(* IEC 61131-3 sources: AOI-sys-for-TI/src/plc, 3 files *)

(* ---- safety_program.st ---- *)
(* ==========================================================================
 * Program:     SAFETY_PROGRAM
 * Description: Safety PLC Logic for AOI Inspection System
 * Target:      Mitsubishi iQ-R Safety CPU (R6SFM)
 * Standard:    ISO 13849-1 PLd, Category 3 (dual-channel with diagnostics)
 *              IEC 62061 SIL 2
 * Notes:       All safety-related I/O uses dual-channel cross-monitoring.
 *              Diagnostic coverage (DC) >= 90% per ISO 13849-1 Table D.2.
 *              CC-Link IE Field Safety protocol for distributed safety I/O.
 * ========================================================================== *)

SAFETY_PROGRAM SAFETY_MAIN

(* ---- Safety I/O Type Definitions ---------------------------------------- *)
TYPE ST_DUAL_CHANNEL : STRUCT
    CH_A             : BOOL;          (* Primary channel input *)
    CH_B             : BOOL;          (* Redundant channel input *)
    DISCREPANCY      : BOOL;          (* Cross-monitor fault detected *)
    DISC_TIMER       : TON;           (* Discrepancy time window *)
    VALID            : BOOL;          (* Both channels agree and healthy *)
END_STRUCT;
END_TYPE

TYPE ST_LIGHT_CURTAIN : STRUCT
    OSSD_1           : BOOL;          (* IEC 61496 Type 2 output 1 *)
    OSSD_2           : BOOL;          (* Redundant safety output 2 *)
    MUTING_ACTIVE    : BOOL;          (* Muting lamp + bypass engaged *)
    BLANKING_ZONE    : USINT;         (* Fixed blanking for material passage *)
    FAULT            : BOOL;
END_STRUCT;
END_TYPE

(* ---- Safety Variables --------------------------------------------------- *)
VAR
    (* E-Stop circuits: 3 buttons per ISO 13850 (twist-release, red/yellow) *)
    ESTOP_1          : ST_DUAL_CHANNEL;   (* Main operator panel *)
    ESTOP_2          : ST_DUAL_CHANNEL;   (* Rear access panel *)
    ESTOP_3          : ST_DUAL_CHANNEL;   (* Teach pendant / mobile *)

    (* Light curtains: IEC 61496 Type 2, 14mm resolution *)
    LC_LOAD_ZONE     : ST_LIGHT_CURTAIN;  (* Loading side *)
    LC_UNLOAD_ZONE   : ST_LIGHT_CURTAIN;  (* Unloading side *)

    (* Safety door interlocks: tongue-type with solenoid lock *)
    DOOR_FRONT       : ST_DUAL_CHANNEL;   (* Front maintenance door *)
    DOOR_REAR        : ST_DUAL_CHANNEL;   (* Rear access door *)
    DOOR_LOCK_FRONT  : BOOL;              (* Solenoid lock output *)
    DOOR_LOCK_REAR   : BOOL;              (* Solenoid lock output *)

    (* Safe Torque Off contactors for servo drives *)
    STO_CONTACTOR_1  : BOOL;              (* Axes 1-4 group *)
    STO_CONTACTOR_2  : BOOL;              (* Axes 5-8 group *)
    STO_FEEDBACK_1   : ST_DUAL_CHANNEL;   (* Contactor weld-check via NC aux *)
    STO_FEEDBACK_2   : ST_DUAL_CHANNEL;

    (* Muting sensors for automatic material handling *)
    MUTE_SENSOR_1    : BOOL;              (* Entry photoeye - conveyor infeed *)
    MUTE_SENSOR_2    : BOOL;              (* Exit photoeye - conveyor infeed *)
    MUTE_SENSOR_3    : BOOL;              (* Entry photoeye - conveyor outfeed *)
    MUTE_SENSOR_4    : BOOL;              (* Exit photoeye - conveyor outfeed *)
    MUTE_TIMER_LOAD  : TON;
    MUTE_TIMER_UNLOAD: TON;

    (* Aggregate outputs *)
    SAFETY_RELAY_OK  : BOOL;              (* Master safety output to main PLC *)
    SAFETY_FAULT_CODE: WORD := 0;
    SAFETY_RESET_PB  : BOOL;              (* Manual reset required after fault *)
    RT_SAFETY_RESET  : R_TRIG;

    (* Discrepancy timing *)
    T_DISC_WINDOW    : TIME := T#500ms;   (* Max allowed discrepancy per Cat.3 *)
    T_MUTE_MAX       : TIME := T#10s;     (* Muting timeout: prevents stuck mute *)

    (* Diagnostic counters -- written to safety log every power cycle *)
    DIAG_ESTOP_TRIPS      : UDINT;
    DIAG_LC_INTERRUPTIONS : UDINT;
    DIAG_DOOR_FAULTS      : UDINT;
    DIAG_DISC_FAULTS      : UDINT;
END_VAR

(* ======================================================================== *)
(* DUAL-CHANNEL CROSS-MONITORING FUNCTION                                   *)
(* Category 3 requires detection of single faults. Discrepancy between      *)
(* channel A and B within T_DISC_WINDOW indicates wiring fault or contact   *)
(* welding. DC >= 90% achieved through cross-monitoring + watchdog.         *)
(* ======================================================================== *)

(* --- E-Stop 1: Main panel ----------------------------------------------- *)
ESTOP_1.DISC_TIMER(IN := (ESTOP_1.CH_A XOR ESTOP_1.CH_B), PT := T_DISC_WINDOW);
ESTOP_1.DISCREPANCY := ESTOP_1.DISC_TIMER.Q;
ESTOP_1.VALID := ESTOP_1.CH_A AND ESTOP_1.CH_B AND NOT ESTOP_1.DISCREPANCY;

(* --- E-Stop 2: Rear panel ----------------------------------------------- *)
ESTOP_2.DISC_TIMER(IN := (ESTOP_2.CH_A XOR ESTOP_2.CH_B), PT := T_DISC_WINDOW);
ESTOP_2.DISCREPANCY := ESTOP_2.DISC_TIMER.Q;
ESTOP_2.VALID := ESTOP_2.CH_A AND ESTOP_2.CH_B AND NOT ESTOP_2.DISCREPANCY;

(* --- E-Stop 3: Mobile / teach pendant ----------------------------------- *)
ESTOP_3.DISC_TIMER(IN := (ESTOP_3.CH_A XOR ESTOP_3.CH_B), PT := T_DISC_WINDOW);
ESTOP_3.DISCREPANCY := ESTOP_3.DISC_TIMER.Q;
ESTOP_3.VALID := ESTOP_3.CH_A AND ESTOP_3.CH_B AND NOT ESTOP_3.DISCREPANCY;

(* --- Light curtain monitoring ------------------------------------------- *)
(* IEC 61496 Type 2: OSSD outputs are antivalent pulsed; both must be TRUE
   for safe condition. Internal diagnostics handled by curtain controller. *)
LC_LOAD_ZONE.FAULT   := (LC_LOAD_ZONE.OSSD_1 XOR LC_LOAD_ZONE.OSSD_2);
LC_UNLOAD_ZONE.FAULT := (LC_UNLOAD_ZONE.OSSD_1 XOR LC_UNLOAD_ZONE.OSSD_2);

(* --- Muting logic for load zone ----------------------------------------- *)
(* Muting allows automatic material (basket/magazine) to pass through the
   light curtain without triggering a safety stop. Sequential activation
   of two cross-beam sensors validates material presence vs. operator.    *)
IF MUTE_SENSOR_1 AND MUTE_SENSOR_2 AND NOT LC_LOAD_ZONE.FAULT THEN
    LC_LOAD_ZONE.MUTING_ACTIVE := TRUE;
    MUTE_TIMER_LOAD(IN := TRUE, PT := T_MUTE_MAX);
ELSE
    IF NOT MUTE_SENSOR_1 AND NOT MUTE_SENSOR_2 THEN
        LC_LOAD_ZONE.MUTING_ACTIVE := FALSE;
        MUTE_TIMER_LOAD(IN := FALSE);
    END_IF;
END_IF;

(* Muting timeout: if material jams, revert to protected mode *)
IF MUTE_TIMER_LOAD.Q THEN
    LC_LOAD_ZONE.MUTING_ACTIVE := FALSE;
    MUTE_TIMER_LOAD(IN := FALSE);
    SAFETY_FAULT_CODE := 16#5001;  (* Muting timeout - check conveyor jam *)
END_IF;

(* --- Muting logic for unload zone --------------------------------------- *)
IF MUTE_SENSOR_3 AND MUTE_SENSOR_4 AND NOT LC_UNLOAD_ZONE.FAULT THEN
    LC_UNLOAD_ZONE.MUTING_ACTIVE := TRUE;
    MUTE_TIMER_UNLOAD(IN := TRUE, PT := T_MUTE_MAX);
ELSE
    IF NOT MUTE_SENSOR_3 AND NOT MUTE_SENSOR_4 THEN
        LC_UNLOAD_ZONE.MUTING_ACTIVE := FALSE;
        MUTE_TIMER_UNLOAD(IN := FALSE);
    END_IF;
END_IF;

IF MUTE_TIMER_UNLOAD.Q THEN
    LC_UNLOAD_ZONE.MUTING_ACTIVE := FALSE;
    MUTE_TIMER_UNLOAD(IN := FALSE);
    SAFETY_FAULT_CODE := 16#5002;
END_IF;

(* --- Safety door interlock monitoring ----------------------------------- *)
DOOR_FRONT.DISC_TIMER(IN := (DOOR_FRONT.CH_A XOR DOOR_FRONT.CH_B), PT := T_DISC_WINDOW);
DOOR_FRONT.DISCREPANCY := DOOR_FRONT.DISC_TIMER.Q;
DOOR_FRONT.VALID := DOOR_FRONT.CH_A AND DOOR_FRONT.CH_B AND NOT DOOR_FRONT.DISCREPANCY;

DOOR_REAR.DISC_TIMER(IN := (DOOR_REAR.CH_A XOR DOOR_REAR.CH_B), PT := T_DISC_WINDOW);
DOOR_REAR.DISCREPANCY := DOOR_REAR.DISC_TIMER.Q;
DOOR_REAR.VALID := DOOR_REAR.CH_A AND DOOR_REAR.CH_B AND NOT DOOR_REAR.DISCREPANCY;

(* Solenoid door locks: keep locked when machine running, unlock on safe stop *)
DOOR_LOCK_FRONT := SAFETY_RELAY_OK;
DOOR_LOCK_REAR  := SAFETY_RELAY_OK;

(* --- STO contactor feedback monitoring ---------------------------------- *)
(* NC auxiliary contacts on STO contactors provide weld-detection.
   If contactor is commanded OFF but feedback shows still ON, weld fault. *)
STO_FEEDBACK_1.DISC_TIMER(IN := (STO_FEEDBACK_1.CH_A XOR STO_FEEDBACK_1.CH_B), PT := T_DISC_WINDOW);
STO_FEEDBACK_1.DISCREPANCY := STO_FEEDBACK_1.DISC_TIMER.Q;
STO_FEEDBACK_1.VALID := STO_FEEDBACK_1.CH_A AND STO_FEEDBACK_1.CH_B AND NOT STO_FEEDBACK_1.DISCREPANCY;

STO_FEEDBACK_2.DISC_TIMER(IN := (STO_FEEDBACK_2.CH_A XOR STO_FEEDBACK_2.CH_B), PT := T_DISC_WINDOW);
STO_FEEDBACK_2.DISCREPANCY := STO_FEEDBACK_2.DISC_TIMER.Q;
STO_FEEDBACK_2.VALID := STO_FEEDBACK_2.CH_A AND STO_FEEDBACK_2.CH_B AND NOT STO_FEEDBACK_2.DISCREPANCY;

(* ======================================================================== *)
(* MASTER SAFETY OUTPUT EVALUATION                                          *)
(* All conditions must be TRUE for machine to operate.                      *)
(* Any single failure -> immediate safe state (STO + pneumatic exhaust).    *)
(*                                                                          *)
(* Diagnostic Coverage Calculation (ISO 13849-1 Table D.4):                 *)
(*   E-Stop dual-channel cross-monitored:        DC = 99%                  *)
(*   Light curtain Type 2 + muting:              DC = 90%                  *)
(*   Safety door interlock dual-channel:         DC = 99%                  *)
(*   STO contactor with weld-check feedback:     DC = 99%                  *)
(*   Overall DC_avg >= 90% -> meets Cat.3 PLd requirement                  *)
(*                                                                          *)
(*   MTTFd per channel > 30 years (high reliability components)            *)
(*   CCF score >= 65 points (separate routing, different manufacturers)     *)
(* ======================================================================== *)

SAFETY_RELAY_OK :=
    ESTOP_1.VALID AND
    ESTOP_2.VALID AND
    ESTOP_3.VALID AND
    DOOR_FRONT.VALID AND
    DOOR_REAR.VALID AND
    (LC_LOAD_ZONE.OSSD_1 AND LC_LOAD_ZONE.OSSD_2 OR LC_LOAD_ZONE.MUTING_ACTIVE) AND
    (LC_UNLOAD_ZONE.OSSD_1 AND LC_UNLOAD_ZONE.OSSD_2 OR LC_UNLOAD_ZONE.MUTING_ACTIVE) AND
    NOT LC_LOAD_ZONE.FAULT AND
    NOT LC_UNLOAD_ZONE.FAULT AND
    STO_FEEDBACK_1.VALID AND
    STO_FEEDBACK_2.VALID AND
    (SAFETY_FAULT_CODE = 0);

(* --- STO contactor control ---------------------------------------------- *)
(* Energise STO contactors only when safety chain is healthy *)
STO_CONTACTOR_1 := SAFETY_RELAY_OK;
STO_CONTACTOR_2 := SAFETY_RELAY_OK;

(* --- Discrepancy fault latching ----------------------------------------- *)
(* Any discrepancy is latched until manual reset per ISO 13849-1 Cat.3     *)
IF ESTOP_1.DISCREPANCY OR ESTOP_2.DISCREPANCY OR ESTOP_3.DISCREPANCY THEN
    SAFETY_FAULT_CODE := 16#E100;  (* E-Stop discrepancy - check wiring *)
    DIAG_DISC_FAULTS := DIAG_DISC_FAULTS + 1;
END_IF;

IF DOOR_FRONT.DISCREPANCY OR DOOR_REAR.DISCREPANCY THEN
    SAFETY_FAULT_CODE := 16#E200;  (* Door interlock discrepancy *)
    DIAG_DOOR_FAULTS := DIAG_DOOR_FAULTS + 1;
END_IF;

IF STO_FEEDBACK_1.DISCREPANCY OR STO_FEEDBACK_2.DISCREPANCY THEN
    SAFETY_FAULT_CODE := 16#E300;  (* STO contactor weld detected *)
    DIAG_DISC_FAULTS := DIAG_DISC_FAULTS + 1;
END_IF;

(* --- Manual reset logic ------------------------------------------------- *)
(* ISO 13849-1 requires monitored manual reset after any safety event.
   Reset button must be outside the hazardous zone.                        *)
RT_SAFETY_RESET(CLK := SAFETY_RESET_PB);
IF RT_SAFETY_RESET.Q THEN
    (* Only allow reset if all physical inputs are in safe state *)
    IF ESTOP_1.CH_A AND ESTOP_1.CH_B AND
       ESTOP_2.CH_A AND ESTOP_2.CH_B AND
       ESTOP_3.CH_A AND ESTOP_3.CH_B AND
       DOOR_FRONT.CH_A AND DOOR_FRONT.CH_B AND
       DOOR_REAR.CH_A AND DOOR_REAR.CH_B THEN
        SAFETY_FAULT_CODE := 0;
    END_IF;
END_IF;

END_PROGRAM

(* ---- main_sequence.st ---- *)
(* =============================================================================
 * Program:     MAIN_SEQUENCE
 * Project:     TI AOI Inspection System
 * Controller:  Mitsubishi iQ-R Series (R16CPU + RJ71GF11-T2)
 * Network:     CC-Link IE Field Basic 1 Gbps (servo + remote I/O)
 *              EtherNet/IP CIP (IPC vision host communication)
 * Cycle Time:  0.5 ms fixed scan | 3.8 s total throughput (4-unit batch)
 * Author:      Controls Engineering
 * Revision:    1.0
 * ========================================================================== *)

PROGRAM MAIN_SEQUENCE

(* ---------------------------------------------------------------------------
 * TYPE DEFINITIONS
 * ------------------------------------------------------------------------ *)
TYPE
    E_INSPECT_STATE : (
        ST_IDLE             := 0,
        ST_BASKET_FEED      := 1,
        ST_CSE_LOAD         := 2,
        ST_PITCH_CHANGE     := 3,
        ST_TRANSFER_1       := 4,
        ST_TRANSFER_2       := 5,
        ST_TRANSFER_3       := 6,
        ST_TRANSFER_4       := 7,
        ST_TRANSFER_5       := 8,
        ST_TRANSFER_6       := 9,
        ST_CCD4_CHECK       := 10,  (* Bottom inspection - inverted optics *)
        ST_CCD3_CHECK       := 11,  (* Top surface inspection *)
        ST_CCD1_CHECK       := 12,  (* Side A + marking verification *)
        ST_ORIENT_COMP      := 13,  (* Theta correction from CCD1 result *)
        ST_CCD2_CHECK       := 14,  (* Side B after orientation alignment *)
        ST_UNLOAD_OK        := 15,
        ST_NG_SORT          := 16,  (* Divert to NG bin by defect class *)
        ST_NG_UNLOAD        := 17,
        ST_ERROR            := 99
    );

    TYPE_VISION_RESULT : STRUCT
        JUDGE           : BOOL;     (* TRUE = PASS, FALSE = NG *)
        DEFECT_CODE     : INT;      (* 0=OK, 1=scratch, 2=chip, 3=mark, 4=foreign *)
        OFFSET_X        : REAL;     (* um, positional deviation *)
        OFFSET_Y        : REAL;
        OFFSET_THETA    : REAL;     (* degrees, rotation deviation *)
        INSPECT_TIME_MS : INT;      (* Vision processing elapsed time *)
    END_STRUCT;

    TYPE_AXIS_CMD : STRUCT
        TARGET_POS      : DINT;     (* Command position in encoder pulses *)
        SPEED           : DINT;     (* mm/s x 100 for fixed-point *)
        ACCEL           : DINT;     (* mm/s^2 x 100 *)
        DECEL           : DINT;
        IN_POSITION     : BOOL;     (* Servo positioning complete feedback *)
        BUSY            : BOOL;
        ERROR           : BOOL;
    END_STRUCT;
END_TYPE

(* ---------------------------------------------------------------------------
 * VARIABLE DECLARATIONS
 * ------------------------------------------------------------------------ *)
VAR
    (* State machine *)
    CURRENT_STATE       : E_INSPECT_STATE := ST_IDLE;
    NEXT_STATE          : E_INSPECT_STATE;
    STATE_ENTRY         : BOOL := TRUE;         (* One-shot on state entry *)
    STEP_TIMER          : TON;                  (* Timeout watchdog per step *)
    CYCLE_TIMER         : TON;                  (* Total cycle time monitor *)
    STEP_TIMEOUT_MS     : TIME := T#5000ms;     (* Max dwell per state *)

    (* CC-Link IE Field cyclic I/O - 8 servo axes *)
    AXIS              : ARRAY[1..8] OF TYPE_AXIS_CMD;
    (* Axis mapping:
       1 = Transfer 1 (basket to pitch change)
       2 = Transfer 2 (pitch change to CCD4)
       3 = Transfer 3 (CCD4 to CCD3)
       4 = Transfer 4 (CCD3 to CCD1)
       5 = Transfer 5 (CCD1 to orient/CCD2)
       6 = Transfer 6 (orient/CCD2 to unload)
       7 = Orientation compensation theta axis
       8 = Side check rotation axis *)

    (* Vision handshake signals - EtherNet/IP CIP implicit messaging *)
    VISION_TRIG         : ARRAY[1..4] OF BOOL;  (* PLC DO -> camera trigger *)
    VISION_BUSY         : ARRAY[1..4] OF BOOL;  (* IPC -> PLC: processing *)
    VISION_DONE         : ARRAY[1..4] OF BOOL;  (* IPC -> PLC: result ready *)
    VISION_RESULT       : ARRAY[1..4] OF TYPE_VISION_RESULT;
    VISION_TRIG_EDGE    : ARRAY[1..4] OF R_TRIG;

    (* Interlock flags - prevent collision between adjacent transfer units *)
    ZONE_CLEAR          : ARRAY[1..8] OF BOOL;  (* TRUE when zone is safe *)
    TRANSFER_ACTIVE     : ARRAY[1..6] OF BOOL;  (* Transfer in motion *)

    (* Sensors via CC-Link IE Field remote I/O *)
    BASKET_PRESENT      : BOOL;     (* Photoelectric sensor at basket feeder *)
    CSE_LOADED          : BOOL;     (* Vacuum sensor confirms unit pickup *)
    PITCH_COMPLETE      : BOOL;     (* Pitch change mechanism settled *)
    PART_AT_CCD4        : BOOL;
    PART_AT_CCD3        : BOOL;
    PART_AT_CCD1        : BOOL;
    PART_AT_CCD2        : BOOL;
    UNLOAD_CLEAR        : BOOL;     (* Unload conveyor not backed up *)
    NG_BIN_FULL         : ARRAY[1..4] OF BOOL;

    (* Pneumatic control - SMC SY3000 solenoids via CC-Link remote I/O *)
    SOL_CSE_VACUUM      : BOOL;     (* Vacuum chuck engage *)
    SOL_PITCH_CLAMP     : BOOL;     (* Pitch change clamp *)
    SOL_TRANSFER_GRIP   : ARRAY[1..6] OF BOOL;  (* Transfer grippers *)
    SOL_ORIENT_CLAMP    : BOOL;
    SOL_UNLOAD_BLOW     : BOOL;     (* Air blow for part release *)
    SOL_NG_DIVERT       : ARRAY[1..4] OF BOOL;  (* NG bin gate selectors *)

    (* Safety inputs *)
    ESTOP_OK            : BOOL;     (* E-Stop circuit healthy *)
    SAFETY_GATE_CLOSED  : BOOL;
    LIGHT_CURTAIN_OK    : BOOL;
    SERVO_STO_RELEASED  : BOOL;     (* STO not active on any drive *)

    (* Edge detection *)
    RT_START            : R_TRIG;
    RT_RESET            : R_TRIG;
    FT_ESTOP            : F_TRIG;   (* Detect E-Stop falling edge *)

    (* Operator interface *)
    CMD_START           : BOOL;
    CMD_RESET           : BOOL;
    CMD_STOP            : BOOL;
    AUTO_MODE           : BOOL;
    CYCLE_RUNNING       : BOOL;

    (* Diagnostics *)
    BATCH_COUNT         : UDINT;
    NG_COUNT            : UDINT;
    CYCLE_TIME_ACTUAL   : TIME;
    LAST_ERROR_CODE     : INT;
    CONSECUTIVE_NG      : INT;      (* Track consecutive NG for alarm *)
    MAX_CONSECUTIVE_NG  : INT := 5; (* Trigger alarm if 5 in a row *)

    (* Internal *)
    i                   : INT;
    ALL_AXES_IDLE       : BOOL;
    ORIENT_CORRECTION   : REAL;     (* Theta offset from CCD1 result *)
END_VAR

(* ---------------------------------------------------------------------------
 * INTERLOCK EVALUATION
 * Adjacent transfer zones must not overlap. Zone N is clear only when
 * the unit in zone N-1 and N+1 are not actively traversing into zone N.
 * This prevents mechanical collision on the linear rail system.
 * ------------------------------------------------------------------------ *)
FOR i := 1 TO 8 DO
    ZONE_CLEAR[i] := TRUE;
END_FOR;

(* Transfer 1 and 2 share a boundary at pitch change station *)
IF TRANSFER_ACTIVE[2] THEN
    ZONE_CLEAR[1] := FALSE;
END_IF;

(* Each adjacent pair interlocked *)
FOR i := 2 TO 5 DO
    IF TRANSFER_ACTIVE[i - 1] OR TRANSFER_ACTIVE[i + 1] THEN
        ZONE_CLEAR[i] := FALSE;
    END_IF;
END_FOR;

IF TRANSFER_ACTIVE[5] THEN
    ZONE_CLEAR[6] := FALSE;
END_IF;

(* ---------------------------------------------------------------------------
 * EDGE DETECTION
 * ------------------------------------------------------------------------ *)
RT_START(CLK := CMD_START);
RT_RESET(CLK := CMD_RESET);
FT_ESTOP(CLK := ESTOP_OK);

(* E-Stop falling edge forces immediate transition to ERROR *)
IF FT_ESTOP.Q THEN
    CURRENT_STATE := ST_ERROR;
    LAST_ERROR_CODE := 9001;    (* E-Stop activated *)
    STATE_ENTRY := TRUE;
END_IF;

(* Safety interlock - block all motion if safety not satisfied *)
IF NOT ESTOP_OK OR NOT SAFETY_GATE_CLOSED OR NOT SERVO_STO_RELEASED THEN
    IF CURRENT_STATE <> ST_IDLE AND CURRENT_STATE <> ST_ERROR THEN
        CURRENT_STATE := ST_ERROR;
        LAST_ERROR_CODE := 9002;    (* Safety interlock violation *)
        STATE_ENTRY := TRUE;
    END_IF;
END_IF;

(* ---------------------------------------------------------------------------
 * STEP TIMEOUT WATCHDOG
 * Any state exceeding STEP_TIMEOUT_MS indicates a jam or sensor failure.
 * ------------------------------------------------------------------------ *)
STEP_TIMER(IN := CYCLE_RUNNING AND (CURRENT_STATE <> ST_IDLE) AND (CURRENT_STATE <> ST_ERROR),
           PT := STEP_TIMEOUT_MS);
IF STEP_TIMER.Q THEN
    CURRENT_STATE := ST_ERROR;
    LAST_ERROR_CODE := 8001;    (* Step timeout *)
    STATE_ENTRY := TRUE;
END_IF;

(* ---------------------------------------------------------------------------
 * MAIN STATE MACHINE
 * Pipeline architecture: multiple batches in flight simultaneously.
 * State machine controls the critical path; non-blocking parallel
 * operations handled by function blocks below.
 * ------------------------------------------------------------------------ *)
CASE CURRENT_STATE OF

    ST_IDLE:
        IF STATE_ENTRY THEN
            CYCLE_RUNNING := FALSE;
            (* De-energize all transfer grippers *)
            FOR i := 1 TO 6 DO
                SOL_TRANSFER_GRIP[i] := FALSE;
                TRANSFER_ACTIVE[i] := FALSE;
            END_FOR;
            STATE_ENTRY := FALSE;
        END_IF;

        IF RT_START.Q AND AUTO_MODE AND ESTOP_OK AND SAFETY_GATE_CLOSED THEN
            CYCLE_RUNNING := TRUE;
            CYCLE_TIMER(IN := FALSE, PT := T#0ms);  (* Reset cycle timer *)
            CURRENT_STATE := ST_BASKET_FEED;
            STATE_ENTRY := TRUE;
        END_IF;

    ST_BASKET_FEED:
        (* Basket feeder indexes next row of 4 units into pick position *)
        IF STATE_ENTRY THEN
            CYCLE_TIMER(IN := TRUE, PT := T#4000ms);
            STEP_TIMER(IN := FALSE, PT := T#0ms);  (* Reset step watchdog *)
            STATE_ENTRY := FALSE;
        END_IF;

        IF BASKET_PRESENT THEN
            CURRENT_STATE := ST_CSE_LOAD;
            STATE_ENTRY := TRUE;
        END_IF;

    ST_CSE_LOAD:
        (* CSE (Component Supply Equipment) picks 4 units with vacuum chuck *)
        IF STATE_ENTRY THEN
            SOL_CSE_VACUUM := TRUE;
            STEP_TIMER(IN := FALSE, PT := T#0ms);
            STATE_ENTRY := FALSE;
        END_IF;

        IF CSE_LOADED THEN
            CURRENT_STATE := ST_PITCH_CHANGE;
            STATE_ENTRY := TRUE;
        END_IF;

    ST_PITCH_CHANGE:
        (* Expand pitch from tray spacing (2.0mm) to inspection spacing (25mm).
           This allows individual access to each unit at vision stations. *)
        IF STATE_ENTRY THEN
            SOL_PITCH_CLAMP := TRUE;
            AXIS[1].TARGET_POS := 50000;  (* 25mm * 2000 pulses/mm *)
            AXIS[1].SPEED := 50000;       (* 500 mm/s *)
            AXIS[1].ACCEL := 200000;      (* 2000 mm/s^2 *)
            STEP_TIMER(IN := FALSE, PT := T#0ms);
            STATE_ENTRY := FALSE;
        END_IF;

        IF PITCH_COMPLETE AND AXIS[1].IN_POSITION THEN
            CURRENT_STATE := ST_TRANSFER_1;
            STATE_ENTRY := TRUE;
        END_IF;

    ST_TRANSFER_1:
        (* Move batch from pitch change to CCD4 bottom inspection station *)
        IF STATE_ENTRY THEN
            IF ZONE_CLEAR[1] THEN
                TRANSFER_ACTIVE[1] := TRUE;
                SOL_TRANSFER_GRIP[1] := TRUE;
                AXIS[1].TARGET_POS := 200000;  (* 100mm travel *)
                STEP_TIMER(IN := FALSE, PT := T#0ms);
                STATE_ENTRY := FALSE;
            END_IF;
        END_IF;

        IF AXIS[1].IN_POSITION AND PART_AT_CCD4 THEN
            SOL_TRANSFER_GRIP[1] := FALSE;
            TRANSFER_ACTIVE[1] := FALSE;
            CURRENT_STATE := ST_CCD4_CHECK;
            STATE_ENTRY := TRUE;
        END_IF;

    ST_CCD4_CHECK:
        (* Bottom inspection: units pass over upward-facing line scan camera.
           Camera 4 triggers on position, captures full bottom surface. *)
        IF STATE_ENTRY THEN
            VISION_TRIG[4] := TRUE;
            STEP_TIMER(IN := FALSE, PT := T#0ms);
            STATE_ENTRY := FALSE;
        END_IF;

        VISION_TRIG_EDGE[4](CLK := VISION_DONE[4]);
        IF VISION_TRIG_EDGE[4].Q THEN
            VISION_TRIG[4] := FALSE;
            IF NOT VISION_RESULT[4].JUDGE THEN
                (* Bottom NG - mark unit but continue pipeline *)
                NG_COUNT := NG_COUNT + 1;
            END_IF;
            CURRENT_STATE := ST_TRANSFER_2;
            STATE_ENTRY := TRUE;
        END_IF;

    ST_TRANSFER_2:
        IF STATE_ENTRY THEN
            IF ZONE_CLEAR[2] THEN
                TRANSFER_ACTIVE[2] := TRUE;
                SOL_TRANSFER_GRIP[2] := TRUE;
                AXIS[2].TARGET_POS := 200000;
                STEP_TIMER(IN := FALSE, PT := T#0ms);
                STATE_ENTRY := FALSE;
            END_IF;
        END_IF;

        IF AXIS[2].IN_POSITION AND PART_AT_CCD3 THEN
            SOL_TRANSFER_GRIP[2] := FALSE;
            TRANSFER_ACTIVE[2] := FALSE;
            CURRENT_STATE := ST_CCD3_CHECK;
            STATE_ENTRY := TRUE;
        END_IF;

    ST_CCD3_CHECK:
        (* Top surface inspection: area scan camera with coaxial lighting.
           Detects scratches, contamination, and marking defects. *)
        IF STATE_ENTRY THEN
            VISION_TRIG[3] := TRUE;
            STEP_TIMER(IN := FALSE, PT := T#0ms);
            STATE_ENTRY := FALSE;
        END_IF;

        VISION_TRIG_EDGE[3](CLK := VISION_DONE[3]);
        IF VISION_TRIG_EDGE[3].Q THEN
            VISION_TRIG[3] := FALSE;
            CURRENT_STATE := ST_TRANSFER_3;
            STATE_ENTRY := TRUE;
        END_IF;

    ST_TRANSFER_3:
        IF STATE_ENTRY THEN
            IF ZONE_CLEAR[3] THEN
                TRANSFER_ACTIVE[3] := TRUE;
                SOL_TRANSFER_GRIP[3] := TRUE;
                AXIS[3].TARGET_POS := 200000;
                STEP_TIMER(IN := FALSE, PT := T#0ms);
                STATE_ENTRY := FALSE;
            END_IF;
        END_IF;

        IF AXIS[3].IN_POSITION AND PART_AT_CCD1 THEN
            SOL_TRANSFER_GRIP[3] := FALSE;
            TRANSFER_ACTIVE[3] := FALSE;
            CURRENT_STATE := ST_CCD1_CHECK;
            STATE_ENTRY := TRUE;
        END_IF;

    ST_CCD1_CHECK:
        (* Side A inspection + marking OCR. Camera 1 also measures angular
           offset for orientation compensation at next station. *)
        IF STATE_ENTRY THEN
            (* Rotate side-check axis to Side A position *)
            AXIS[8].TARGET_POS := 0;  (* 0 degrees *)
            VISION_TRIG[1] := TRUE;
            STEP_TIMER(IN := FALSE, PT := T#0ms);
            STATE_ENTRY := FALSE;
        END_IF;

        VISION_TRIG_EDGE[1](CLK := VISION_DONE[1]);
        IF VISION_TRIG_EDGE[1].Q THEN
            VISION_TRIG[1] := FALSE;
            (* Capture theta offset for orientation compensation *)
            ORIENT_CORRECTION := VISION_RESULT[1].OFFSET_THETA;
            CURRENT_STATE := ST_TRANSFER_4;
            STATE_ENTRY := TRUE;
        END_IF;

    ST_TRANSFER_4:
        IF STATE_ENTRY THEN
            IF ZONE_CLEAR[4] THEN
                TRANSFER_ACTIVE[4] := TRUE;
                SOL_TRANSFER_GRIP[4] := TRUE;
                AXIS[4].TARGET_POS := 200000;
                STEP_TIMER(IN := FALSE, PT := T#0ms);
                STATE_ENTRY := FALSE;
            END_IF;
        END_IF;

        IF AXIS[4].IN_POSITION THEN
            SOL_TRANSFER_GRIP[4] := FALSE;
            TRANSFER_ACTIVE[4] := FALSE;
            CURRENT_STATE := ST_ORIENT_COMP;
            STATE_ENTRY := TRUE;
        END_IF;

    ST_ORIENT_COMP:
        (* Theta axis corrects angular misalignment measured by CCD1.
           Compensation ensures CCD2 side B image is rotationally aligned. *)
        IF STATE_ENTRY THEN
            SOL_ORIENT_CLAMP := TRUE;
            (* Convert degrees to encoder pulses: 1 deg = 1000 pulses *)
            AXIS[7].TARGET_POS := REAL_TO_DINT(ORIENT_CORRECTION * 1000.0);
            AXIS[7].SPEED := 36000;     (* 360 deg/s *)
            AXIS[7].ACCEL := 720000;    (* Fast settle for throughput *)
            STEP_TIMER(IN := FALSE, PT := T#0ms);
            STATE_ENTRY := FALSE;
        END_IF;

        IF AXIS[7].IN_POSITION THEN
            CURRENT_STATE := ST_CCD2_CHECK;
            STATE_ENTRY := TRUE;
        END_IF;

    ST_CCD2_CHECK:
        (* Side B inspection after orientation alignment *)
        IF STATE_ENTRY THEN
            VISION_TRIG[2] := TRUE;
            STEP_TIMER(IN := FALSE, PT := T#0ms);
            STATE_ENTRY := FALSE;
        END_IF;

        VISION_TRIG_EDGE[2](CLK := VISION_DONE[2]);
        IF VISION_TRIG_EDGE[2].Q THEN
            VISION_TRIG[2] := FALSE;
            SOL_ORIENT_CLAMP := FALSE;
            (* Aggregate all 4 camera results for final judgment *)
            IF VISION_RESULT[1].JUDGE AND VISION_RESULT[2].JUDGE
               AND VISION_RESULT[3].JUDGE AND VISION_RESULT[4].JUDGE THEN
                CURRENT_STATE := ST_TRANSFER_5;
            ELSE
                CURRENT_STATE := ST_NG_SORT;
            END_IF;
            STATE_ENTRY := TRUE;
        END_IF;

    ST_TRANSFER_5:
        (* Move passed units to OK unload station *)
        IF STATE_ENTRY THEN
            IF ZONE_CLEAR[5] THEN
                TRANSFER_ACTIVE[5] := TRUE;
                SOL_TRANSFER_GRIP[5] := TRUE;
                AXIS[5].TARGET_POS := 200000;
                STEP_TIMER(IN := FALSE, PT := T#0ms);
                STATE_ENTRY := FALSE;
            END_IF;
        END_IF;

        IF AXIS[5].IN_POSITION THEN
            SOL_TRANSFER_GRIP[5] := FALSE;
            TRANSFER_ACTIVE[5] := FALSE;
            CURRENT_STATE := ST_UNLOAD_OK;
            STATE_ENTRY := TRUE;
        END_IF;

    ST_UNLOAD_OK:
        (* Release passed units onto OK conveyor via air blow *)
        IF STATE_ENTRY THEN
            SOL_UNLOAD_BLOW := TRUE;
            STEP_TIMER(IN := FALSE, PT := T#0ms);
            STATE_ENTRY := FALSE;
        END_IF;

        IF UNLOAD_CLEAR THEN
            SOL_UNLOAD_BLOW := FALSE;
            BATCH_COUNT := BATCH_COUNT + 1;
            CONSECUTIVE_NG := 0;
            CURRENT_STATE := ST_IDLE;
            STATE_ENTRY := TRUE;
        END_IF;

    ST_NG_SORT:
        (* Route NG units to appropriate bin based on defect classification.
           Bins: 1=scratch, 2=chip, 3=marking, 4=foreign/other *)
        IF STATE_ENTRY THEN
            IF ZONE_CLEAR[6] THEN
                TRANSFER_ACTIVE[6] := TRUE;
                SOL_TRANSFER_GRIP[6] := TRUE;
                (* Determine NG bin from worst defect code across all cameras *)
                FOR i := 1 TO 4 DO
                    IF NOT VISION_RESULT[i].JUDGE AND VISION_RESULT[i].DEFECT_CODE > 0
                       AND VISION_RESULT[i].DEFECT_CODE <= 4 THEN
                        SOL_NG_DIVERT[VISION_RESULT[i].DEFECT_CODE] := TRUE;
                    END_IF;
                END_FOR;
                STEP_TIMER(IN := FALSE, PT := T#0ms);
                STATE_ENTRY := FALSE;
            END_IF;
        END_IF;

        IF AXIS[6].IN_POSITION THEN
            CURRENT_STATE := ST_NG_UNLOAD;
            STATE_ENTRY := TRUE;
        END_IF;

    ST_NG_UNLOAD:
        IF STATE_ENTRY THEN
            SOL_TRANSFER_GRIP[6] := FALSE;
            TRANSFER_ACTIVE[6] := FALSE;
            STEP_TIMER(IN := FALSE, PT := T#0ms);
            STATE_ENTRY := FALSE;
        END_IF;

        (* Wait for NG unit to clear the divert gate sensor *)
        IF NOT PART_AT_CCD2 THEN
            FOR i := 1 TO 4 DO
                SOL_NG_DIVERT[i] := FALSE;
            END_FOR;
            NG_COUNT := NG_COUNT + 1;
            CONSECUTIVE_NG := CONSECUTIVE_NG + 1;
            IF CONSECUTIVE_NG >= MAX_CONSECUTIVE_NG THEN
                CURRENT_STATE := ST_ERROR;
                LAST_ERROR_CODE := 7001;  (* Consecutive NG alarm *)
                STATE_ENTRY := TRUE;
            ELSE
                CURRENT_STATE := ST_IDLE;
                STATE_ENTRY := TRUE;
            END_IF;
        END_IF;

    ST_ERROR:
        IF STATE_ENTRY THEN
            (* Immediate safe shutdown: release all grippers, disable servos *)
            FOR i := 1 TO 6 DO
                SOL_TRANSFER_GRIP[i] := FALSE;
                TRANSFER_ACTIVE[i] := FALSE;
            END_FOR;
            SOL_CSE_VACUUM := FALSE;
            SOL_ORIENT_CLAMP := FALSE;
            SOL_UNLOAD_BLOW := FALSE;
            CYCLE_RUNNING := FALSE;
            STATE_ENTRY := FALSE;
        END_IF;

        (* Operator must acknowledge error and press reset *)
        IF RT_RESET.Q AND ESTOP_OK AND SAFETY_GATE_CLOSED THEN
            LAST_ERROR_CODE := 0;
            CONSECUTIVE_NG := 0;
            CURRENT_STATE := ST_IDLE;
            STATE_ENTRY := TRUE;
        END_IF;

END_CASE;

(* ---------------------------------------------------------------------------
 * CYCLE TIME MEASUREMENT
 * Record actual cycle time for OEE calculation. Target: 3.8s per batch.
 * Alarm if sustained above 4.2s (>10% degradation).
 * ------------------------------------------------------------------------ *)
IF CURRENT_STATE = ST_IDLE AND CYCLE_RUNNING = FALSE THEN
    CYCLE_TIME_ACTUAL := CYCLE_TIMER.ET;
END_IF;

(* ---------------------------------------------------------------------------
 * VISION HANDSHAKE MONITOR
 * EtherNet/IP CIP connection watchdog. If IPC does not respond within
 * 500ms of trigger, assume communication fault.
 * ------------------------------------------------------------------------ *)
FOR i := 1 TO 4 DO
    IF VISION_TRIG[i] AND NOT VISION_BUSY[i] AND NOT VISION_DONE[i] THEN
        (* Trigger sent, waiting for IPC acknowledgment *)
        (* Timeout handled by STEP_TIMER at state level *)
    END_IF;
END_FOR;

END_PROGRAM

(* ---- servo_config.st ---- *)
(* ==========================================================================
 * Program:     SERVO_CONFIG
 * Description: 8-Axis Servo Drive Configuration and Homing Sequences
 * Drives:      Mitsubishi MR-J5-G series via CC-Link IE Field
 * Network:     CC-Link IE Field 1 Gbps, 0.5 ms communication cycle
 * Motion:      Position mode (CP), electronic gear via drive parameters
 * ========================================================================== *)

PROGRAM SERVO_CONFIG

(* ---- Axis Configuration Type ------------------------------------------- *)
TYPE ST_AXIS_CONFIG : STRUCT
    AXIS_NAME        : STRING[32];
    MOTION_TYPE      : USINT;        (* 0=Linear [mm], 1=Rotary [deg] *)
    GEAR_NUM         : UDINT;        (* Electronic gear numerator *)
    GEAR_DEN         : UDINT;        (* Electronic gear denominator *)
    ENCODER_PPR      : UDINT;        (* Encoder pulses per revolution *)
    BALL_SCREW_LEAD  : LREAL;        (* [mm/rev], 0 for direct-drive rotary *)
    MAX_VELOCITY     : LREAL;        (* [mm/s] or [deg/s] *)
    MAX_ACCEL        : LREAL;        (* [mm/s^2] or [deg/s^2] *)
    MAX_DECEL        : LREAL;
    JOG_VELOCITY     : LREAL;        (* Manual jog speed *)
    HOME_VELOCITY    : LREAL;        (* Homing approach speed *)
    HOME_CREEP       : LREAL;        (* Slow final approach to home sensor *)
    HOME_OFFSET      : LREAL;        (* Distance from home sensor to datum *)
    HOME_DIRECTION   : BOOL;         (* FALSE=negative, TRUE=positive *)
    SW_LIMIT_POS     : LREAL;        (* Software positive limit *)
    SW_LIMIT_NEG     : LREAL;        (* Software negative limit *)
    IN_POS_BAND      : LREAL;        (* In-position tolerance band *)
    TORQUE_LIMIT     : LREAL;        (* [%] of rated torque *)
END_STRUCT;
END_TYPE

TYPE ST_AXIS_STATUS : STRUCT
    ACTUAL_POS       : LREAL;
    ACTUAL_VEL       : LREAL;
    ACTUAL_TORQUE    : LREAL;        (* [%] of rated *)
    IS_HOMED         : BOOL;
    IS_ENABLED       : BOOL;
    IS_MOVING        : BOOL;
    IS_IN_POSITION   : BOOL;
    ALARM_CODE       : WORD;
    ALARM_HISTORY    : ARRAY[0..7] OF WORD;  (* Last 8 alarms for diagnostics *)
END_STRUCT;
END_TYPE

(* ---- Homing State Machine ---------------------------------------------- *)
TYPE E_HOME_STATE : (
    HOME_IDLE        := 0,
    HOME_SEEK_SWITCH := 1,       (* Fast approach toward home sensor *)
    HOME_BACK_OFF    := 2,       (* Reverse off sensor at creep speed *)
    HOME_FINAL_APP   := 3,       (* Final slow approach to sensor edge *)
    HOME_SET_ORIGIN  := 4,       (* Capture position, apply offset *)
    HOME_COMPLETE    := 5,
    HOME_ERROR       := 99
);
END_TYPE

(* ---- Variables --------------------------------------------------------- *)
VAR
    AXIS_CFG         : ARRAY[1..8] OF ST_AXIS_CONFIG;
    AXIS_STAT        : ARRAY[1..8] OF ST_AXIS_STATUS;
    HOME_STATE       : ARRAY[1..8] OF E_HOME_STATE;
    HOME_REQUEST     : BOOL;           (* Triggers all-axis homing sequence *)
    HOME_AXIS_INDEX  : USINT := 1;     (* Sequential homing: one axis at a time *)
    ALL_AXES_HOMED   : BOOL;
    HOME_TIMER       : TON;
    RT_HOME_REQ      : R_TRIG;
    i                : INT;
END_VAR

VAR CONSTANT
    T_HOME_TIMEOUT   : TIME := T#30s;  (* Per-axis homing timeout *)
END_VAR

(* ======================================================================== *)
(* AXIS PARAMETER INITIALIZATION                                            *)
(* Run once on first scan or after parameter download from HMI              *)
(* Electronic gear: (GEAR_NUM / GEAR_DEN) * ENCODER_PPR = pulses per mm     *)
(* ======================================================================== *)

(* --- Axis 1: Transfer 1 (basket -> CSE loader) --- *)
(* Mitsubishi HK-KT23W, 200W, ball screw driven linear slide *)
AXIS_CFG[1].AXIS_NAME       := 'TRANSFER_1';
AXIS_CFG[1].MOTION_TYPE     := 0;          (* Linear *)
AXIS_CFG[1].GEAR_NUM        := 1;
AXIS_CFG[1].GEAR_DEN        := 1;
AXIS_CFG[1].ENCODER_PPR     := 4194304;    (* 22-bit absolute encoder *)
AXIS_CFG[1].BALL_SCREW_LEAD := 10.0;       (* 10 mm/rev C5 precision *)
AXIS_CFG[1].MAX_VELOCITY    := 1000.0;     (* mm/s *)
AXIS_CFG[1].MAX_ACCEL       := 10000.0;    (* mm/s^2, ~1G *)
AXIS_CFG[1].MAX_DECEL       := 10000.0;
AXIS_CFG[1].JOG_VELOCITY    := 50.0;
AXIS_CFG[1].HOME_VELOCITY   := 100.0;
AXIS_CFG[1].HOME_CREEP      := 5.0;
AXIS_CFG[1].HOME_OFFSET     := 2.0;
AXIS_CFG[1].HOME_DIRECTION  := FALSE;      (* Home toward negative limit *)
AXIS_CFG[1].SW_LIMIT_POS    := 200.0;
AXIS_CFG[1].SW_LIMIT_NEG    := -1.0;
AXIS_CFG[1].IN_POS_BAND     := 0.005;      (* 5 um *)
AXIS_CFG[1].TORQUE_LIMIT    := 100.0;

(* --- Axis 2: Transfer 2 (CSE -> pitch change) --- *)
AXIS_CFG[2].AXIS_NAME       := 'TRANSFER_2';
AXIS_CFG[2].MOTION_TYPE     := 0;
AXIS_CFG[2].GEAR_NUM        := 1;
AXIS_CFG[2].GEAR_DEN        := 1;
AXIS_CFG[2].ENCODER_PPR     := 4194304;
AXIS_CFG[2].BALL_SCREW_LEAD := 10.0;
AXIS_CFG[2].MAX_VELOCITY    := 1000.0;
AXIS_CFG[2].MAX_ACCEL       := 10000.0;
AXIS_CFG[2].MAX_DECEL       := 10000.0;
AXIS_CFG[2].JOG_VELOCITY    := 50.0;
AXIS_CFG[2].HOME_VELOCITY   := 100.0;
AXIS_CFG[2].HOME_CREEP      := 5.0;
AXIS_CFG[2].HOME_OFFSET     := 2.0;
AXIS_CFG[2].HOME_DIRECTION  := FALSE;
AXIS_CFG[2].SW_LIMIT_POS    := 250.0;
AXIS_CFG[2].SW_LIMIT_NEG    := -1.0;
AXIS_CFG[2].IN_POS_BAND     := 0.005;
AXIS_CFG[2].TORQUE_LIMIT    := 100.0;

(* --- Axis 3: Transfer 3 (pitch change -> CCD4) --- *)
AXIS_CFG[3].AXIS_NAME       := 'TRANSFER_3';
AXIS_CFG[3].MOTION_TYPE     := 0;
AXIS_CFG[3].GEAR_NUM        := 1;
AXIS_CFG[3].GEAR_DEN        := 1;
AXIS_CFG[3].ENCODER_PPR     := 4194304;
AXIS_CFG[3].BALL_SCREW_LEAD := 10.0;
AXIS_CFG[3].MAX_VELOCITY    := 1200.0;     (* Faster: longer travel *)
AXIS_CFG[3].MAX_ACCEL       := 12000.0;
AXIS_CFG[3].MAX_DECEL       := 12000.0;
AXIS_CFG[3].JOG_VELOCITY    := 50.0;
AXIS_CFG[3].HOME_VELOCITY   := 100.0;
AXIS_CFG[3].HOME_CREEP      := 5.0;
AXIS_CFG[3].HOME_OFFSET     := 2.0;
AXIS_CFG[3].HOME_DIRECTION  := FALSE;
AXIS_CFG[3].SW_LIMIT_POS    := 500.0;
AXIS_CFG[3].SW_LIMIT_NEG    := -1.0;
AXIS_CFG[3].IN_POS_BAND     := 0.005;
AXIS_CFG[3].TORQUE_LIMIT    := 100.0;

(* --- Axis 4: Transfer 4 (CCD4 -> CCD3) --- *)
AXIS_CFG[4].AXIS_NAME       := 'TRANSFER_4';
AXIS_CFG[4].MOTION_TYPE     := 0;
AXIS_CFG[4].GEAR_NUM        := 1;
AXIS_CFG[4].GEAR_DEN        := 1;
AXIS_CFG[4].ENCODER_PPR     := 4194304;
AXIS_CFG[4].BALL_SCREW_LEAD := 10.0;
AXIS_CFG[4].MAX_VELOCITY    := 1200.0;
AXIS_CFG[4].MAX_ACCEL       := 12000.0;
AXIS_CFG[4].MAX_DECEL       := 12000.0;
AXIS_CFG[4].JOG_VELOCITY    := 50.0;
AXIS_CFG[4].HOME_VELOCITY   := 100.0;
AXIS_CFG[4].HOME_CREEP      := 5.0;
AXIS_CFG[4].HOME_OFFSET     := 2.0;
AXIS_CFG[4].HOME_DIRECTION  := FALSE;
AXIS_CFG[4].SW_LIMIT_POS    := 500.0;
AXIS_CFG[4].SW_LIMIT_NEG    := -1.0;
AXIS_CFG[4].IN_POS_BAND     := 0.005;
AXIS_CFG[4].TORQUE_LIMIT    := 100.0;

(* --- Axis 5: Transfer 5 (CCD3 -> CCD1/orientation) --- *)
AXIS_CFG[5].AXIS_NAME       := 'TRANSFER_5';
AXIS_CFG[5].MOTION_TYPE     := 0;
AXIS_CFG[5].GEAR_NUM        := 1;
AXIS_CFG[5].GEAR_DEN        := 1;
AXIS_CFG[5].ENCODER_PPR     := 4194304;
AXIS_CFG[5].BALL_SCREW_LEAD := 10.0;
AXIS_CFG[5].MAX_VELOCITY    := 800.0;      (* Slower: precision placement *)
AXIS_CFG[5].MAX_ACCEL       := 8000.0;
AXIS_CFG[5].MAX_DECEL       := 8000.0;
AXIS_CFG[5].JOG_VELOCITY    := 30.0;
AXIS_CFG[5].HOME_VELOCITY   := 80.0;
AXIS_CFG[5].HOME_CREEP      := 3.0;
AXIS_CFG[5].HOME_OFFSET     := 2.0;
AXIS_CFG[5].HOME_DIRECTION  := FALSE;
AXIS_CFG[5].SW_LIMIT_POS    := 800.0;
AXIS_CFG[5].SW_LIMIT_NEG    := -1.0;
AXIS_CFG[5].IN_POS_BAND     := 0.003;      (* Tighter: orientation station *)
AXIS_CFG[5].TORQUE_LIMIT    := 80.0;

(* --- Axis 6: Transfer 6 (CCD2 -> unload) --- *)
AXIS_CFG[6].AXIS_NAME       := 'TRANSFER_6';
AXIS_CFG[6].MOTION_TYPE     := 0;
AXIS_CFG[6].GEAR_NUM        := 1;
AXIS_CFG[6].GEAR_DEN        := 1;
AXIS_CFG[6].ENCODER_PPR     := 4194304;
AXIS_CFG[6].BALL_SCREW_LEAD := 10.0;
AXIS_CFG[6].MAX_VELOCITY    := 1000.0;
AXIS_CFG[6].MAX_ACCEL       := 10000.0;
AXIS_CFG[6].MAX_DECEL       := 10000.0;
AXIS_CFG[6].JOG_VELOCITY    := 50.0;
AXIS_CFG[6].HOME_VELOCITY   := 100.0;
AXIS_CFG[6].HOME_CREEP      := 5.0;
AXIS_CFG[6].HOME_OFFSET     := 2.0;
AXIS_CFG[6].HOME_DIRECTION  := FALSE;
AXIS_CFG[6].SW_LIMIT_POS    := 950.0;
AXIS_CFG[6].SW_LIMIT_NEG    := -1.0;
AXIS_CFG[6].IN_POS_BAND     := 0.005;
AXIS_CFG[6].TORQUE_LIMIT    := 100.0;

(* --- Axis 7: Orientation Compensation (rotary, direct-drive) --- *)
(* Mitsubishi HK-KT13, 100W, direct-drive rotary table *)
AXIS_CFG[7].AXIS_NAME       := 'ORIENT_COMP';
AXIS_CFG[7].MOTION_TYPE     := 1;          (* Rotary *)
AXIS_CFG[7].GEAR_NUM        := 1;
AXIS_CFG[7].GEAR_DEN        := 72;         (* 72:1 harmonic drive reduction *)
AXIS_CFG[7].ENCODER_PPR     := 4194304;
AXIS_CFG[7].BALL_SCREW_LEAD := 0.0;        (* N/A for rotary *)
AXIS_CFG[7].MAX_VELOCITY    := 360.0;      (* deg/s *)
AXIS_CFG[7].MAX_ACCEL       := 3600.0;     (* deg/s^2 *)
AXIS_CFG[7].MAX_DECEL       := 3600.0;
AXIS_CFG[7].JOG_VELOCITY    := 10.0;
AXIS_CFG[7].HOME_VELOCITY   := 30.0;
AXIS_CFG[7].HOME_CREEP      := 2.0;
AXIS_CFG[7].HOME_OFFSET     := 0.0;
AXIS_CFG[7].HOME_DIRECTION  := TRUE;       (* Home toward positive/CW *)
AXIS_CFG[7].SW_LIMIT_POS    := 180.0;      (* +/- 180 deg range *)
AXIS_CFG[7].SW_LIMIT_NEG    := -180.0;
AXIS_CFG[7].IN_POS_BAND     := 0.01;       (* 0.01 deg = 36 arcsec *)
AXIS_CFG[7].TORQUE_LIMIT    := 50.0;       (* Low inertia load *)

(* --- Axis 8: CCD3 Side-Check 360-deg Rotation --- *)
(* Mitsubishi HK-KT23W, 200W, direct-drive continuous rotation *)
AXIS_CFG[8].AXIS_NAME       := 'SIDE_CHECK_ROT';
AXIS_CFG[8].MOTION_TYPE     := 1;          (* Rotary *)
AXIS_CFG[8].GEAR_NUM        := 1;
AXIS_CFG[8].GEAR_DEN        := 50;         (* 50:1 worm gear for backlash-free *)
AXIS_CFG[8].ENCODER_PPR     := 4194304;
AXIS_CFG[8].BALL_SCREW_LEAD := 0.0;
AXIS_CFG[8].MAX_VELOCITY    := 1080.0;     (* deg/s - 3 rev/s max *)
AXIS_CFG[8].MAX_ACCEL       := 7200.0;
AXIS_CFG[8].MAX_DECEL       := 7200.0;
AXIS_CFG[8].JOG_VELOCITY    := 30.0;
AXIS_CFG[8].HOME_VELOCITY   := 60.0;
AXIS_CFG[8].HOME_CREEP      := 5.0;
AXIS_CFG[8].HOME_OFFSET     := 0.0;
AXIS_CFG[8].HOME_DIRECTION  := TRUE;
AXIS_CFG[8].SW_LIMIT_POS    := 99999.0;    (* No limit: continuous rotation *)
AXIS_CFG[8].SW_LIMIT_NEG    := -99999.0;
AXIS_CFG[8].IN_POS_BAND     := 0.05;       (* Relaxed: full-revolution scan *)
AXIS_CFG[8].TORQUE_LIMIT    := 80.0;

(* ======================================================================== *)
(* HOMING SEQUENCE STATE MACHINE                                            *)
(* Sequential homing: axes home one at a time to prevent collision.          *)
(* Order: 7 (orient) -> 8 (rotation) -> 1 -> 2 -> 3 -> 4 -> 5 -> 6        *)
(* Rotary axes home first as they have no collision risk with linear axes.  *)
(* ======================================================================== *)

VAR CONSTANT
    HOME_ORDER : ARRAY[1..8] OF USINT := [7, 8, 1, 2, 3, 4, 5, 6];
END_VAR

RT_HOME_REQ(CLK := HOME_REQUEST);
IF RT_HOME_REQ.Q THEN
    HOME_AXIS_INDEX := 1;
    FOR i := 1 TO 8 DO
        HOME_STATE[i] := HOME_IDLE;
        AXIS_STAT[i].IS_HOMED := FALSE;
    END_FOR;
END_IF;

(* Process current homing axis *)
IF HOME_AXIS_INDEX >= 1 AND HOME_AXIS_INDEX <= 8 THEN

    CASE HOME_STATE[HOME_ORDER[HOME_AXIS_INDEX]] OF

        HOME_IDLE:
            (* Initiate homing for current axis in sequence *)
            IF HOME_REQUEST THEN
                HOME_STATE[HOME_ORDER[HOME_AXIS_INDEX]] := HOME_SEEK_SWITCH;
                HOME_TIMER(IN := FALSE);  (* Reset timeout *)
            END_IF;

        HOME_SEEK_SWITCH:
            (* Fast approach toward home sensor *)
            (* Velocity = HOME_VELOCITY in configured HOME_DIRECTION *)
            HOME_TIMER(IN := TRUE, PT := T_HOME_TIMEOUT);

            (* Simulated: in real system, motion command issued to drive via
               CC-Link IE Field parameter Pr.52 (home mode), Pr.53 (home speed).
               Drive handles the physical motion; PLC monitors completion. *)

            IF AXIS_STAT[HOME_ORDER[HOME_AXIS_INDEX]].IS_IN_POSITION THEN
                HOME_STATE[HOME_ORDER[HOME_AXIS_INDEX]] := HOME_BACK_OFF;
            END_IF;

            IF HOME_TIMER.Q THEN
                HOME_STATE[HOME_ORDER[HOME_AXIS_INDEX]] := HOME_ERROR;
            END_IF;

        HOME_BACK_OFF:
            (* Reverse direction at creep speed to back off home sensor *)
            (* This gives a clean edge detection on second approach *)
            HOME_STATE[HOME_ORDER[HOME_AXIS_INDEX]] := HOME_FINAL_APP;

        HOME_FINAL_APP:
            (* Final slow approach to home sensor rising edge *)
            (* Drive captures encoder position at sensor transition *)
            IF AXIS_STAT[HOME_ORDER[HOME_AXIS_INDEX]].IS_IN_POSITION THEN
                HOME_STATE[HOME_ORDER[HOME_AXIS_INDEX]] := HOME_SET_ORIGIN;
            END_IF;

        HOME_SET_ORIGIN:
            (* Apply home offset: datum = sensor_pos + HOME_OFFSET *)
            (* Write absolute position origin via CC-Link IE Field Pr.901 *)
            AXIS_STAT[HOME_ORDER[HOME_AXIS_INDEX]].IS_HOMED := TRUE;
            AXIS_STAT[HOME_ORDER[HOME_AXIS_INDEX]].ACTUAL_POS := 0.0;
            HOME_STATE[HOME_ORDER[HOME_AXIS_INDEX]] := HOME_COMPLETE;

        HOME_COMPLETE:
            (* Advance to next axis in homing order *)
            HOME_TIMER(IN := FALSE);
            IF HOME_AXIS_INDEX < 8 THEN
                HOME_AXIS_INDEX := HOME_AXIS_INDEX + 1;
                HOME_STATE[HOME_ORDER[HOME_AXIS_INDEX]] := HOME_SEEK_SWITCH;
            END_IF;

        HOME_ERROR:
            (* Homing failed: alarm and halt sequence *)
            (* Operator must resolve obstruction and re-request homing *)
            HOME_TIMER(IN := FALSE);
            HOME_REQUEST := FALSE;

    END_CASE;

END_IF;

(* --- Aggregate homed status --------------------------------------------- *)
ALL_AXES_HOMED := TRUE;
FOR i := 1 TO 8 DO
    IF NOT AXIS_STAT[i].IS_HOMED THEN
        ALL_AXES_HOMED := FALSE;
    END_IF;
END_FOR;

(* ======================================================================== *)
(* CC-LINK IE FIELD SERVO PARAMETER MAPPING                                 *)
(* MR-J5-G drive parameters mapped to cyclic communication buffer           *)
(*                                                                          *)
(* Cyclic Transmission (RWw/RWr):                                           *)
(*   RWw0: Control word (servo ON, start, stop, home)                       *)
(*   RWw1-RWw2: Target position [pulse] (32-bit)                            *)
(*   RWw3: Target velocity [rpm]                                            *)
(*   RWw4: Acceleration time [ms]                                           *)
(*   RWw5: Deceleration time [ms]                                           *)
(*   RWr0: Status word (ready, in-position, alarm, homed)                   *)
(*   RWr1-RWr2: Actual position [pulse] (32-bit)                            *)
(*   RWr3: Actual velocity [rpm]                                            *)
(*   RWr4: Actual torque [0.1%]                                             *)
(*   RWr5: Alarm code                                                       *)
(*                                                                          *)
(* Station assignment (CC-Link IE Field):                                   *)
(*   Station 2, Slots 0-1: Axes 1-4 (transfer drives)                      *)
(*   Station 3, Slots 0-1: Axes 5-8 (transfer + rotary drives)             *)
(* ======================================================================== *)

END_PROGRAM
